// TwinCAT 3 PLC project testPLC
// ProgramVersion: 3.1.4026.1+c9eadab3edd020c56c333d811d5b3c408c2550c8
// libraries:
//   Tc2_Standard, * (Beckhoff Automation GmbH)
//   Tc2_System, * (Beckhoff Automation GmbH)
// project tree:
//   / PlcTask.TcTTO
//   POUs/ FB_Generics.TcPOU, FB_Methods.TcPOU, MAIN.TcPOU
// real-time tasks:
//   TASK PlcTask: cycle T#10ms, priority 20, ADS port 350

CONFIGURATION testPLC
    RESOURCE PLC ON TwinCAT3
        TASK PlcTask(INTERVAL := T#10ms, PRIORITY := 20);
        PROGRAM MAIN WITH PlcTask : MAIN;
    END_RESOURCE
END_CONFIGURATION

// ---- POUs/MAIN.TcPOU
PROGRAM MAIN
VAR
	testMethods		: FB_Methods;
	testGenerics	: FB_Generics<100>;
END_VAR

testMethods.MethodDefaultValue(1);

END_PROGRAM

// ---- POUs/FB_Methods.TcPOU
FUNCTION_BLOCK FB_Methods
VAR 
	
END_VAR

METHOD MethodDefaultValue
VAR_INPUT
	nValue1		: INT;
	nValue2		: INT := 5;
END_VAR
END_METHOD

END_FUNCTION_BLOCK

// ---- POUs/FB_Generics.TcPOU
FUNCTION_BLOCK FB_Generics
VAR_GENERIC CONSTANT
	nArraySize 	: INT := 10;
END_VAR
VAR 
	nStrArray	: ARRAY[0..nArraySize] OF STRING(255);
END_VAR

END_FUNCTION_BLOCK
